{attribute 'qualified_only'}
VAR_GLOBAL PERSISTENT //to be persistent
	MyPersistentInteger : INT := 10;
END_VAR

VAR_GLOBAL // non persistent
	MyNonPersistentInteger : INT :=10;
END_VAR

(* stored: Version 1.1.0.1, ProductVersion 3.1.4020.12
   GVL PersistentExample: Id {cfde9f39-e1f2-4403-8a96-556ac735df51} *)
